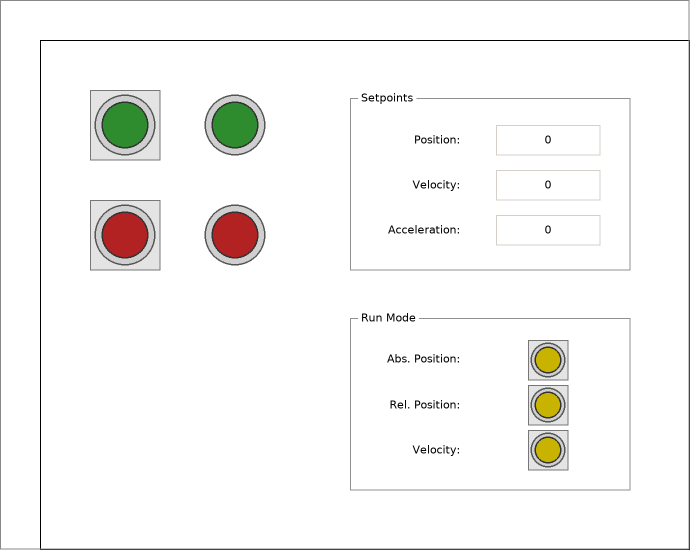
VISUALIZATION Visualization  // 690x550
    RoundedRectangle (40,40 650x510)
    PushSwitch (90,90 70x70), tooltip "START", behaviour: TOGGLE, style: Switch-PushSwitch-Green
    Lamp1 (200,90 70x70), style: Lamp-Lamp1-Green
    PushSwitch (90,200 70x70), tooltip "STOP", behaviour: TOGGLE, style: Switch-PushSwitch-Red
    Lamp1 (200,200 70x70), style: Lamp-Lamp1-Red
    GroupBox (350,90 280x180), "Setpoints"
        Label (16,80 97x30), "Velocity:"
        Label (16,125 97x30), "Acceleration:"
        Textfield (146,80 104x30), "0"
        Textfield (146,35 104x30), "0"
        Textfield (146,125 104x30), "0"
        Label (16,35 97x30), "Position:"
    GroupBox (350,310 280x180), "Run Mode"
        Label (16,80 97x30), "Rel. Position:"
        Label (16,125 97x30), "Velocity:"
        Label (16,34 97x30), "Abs. Position:"
        PushSwitch (178,30 40x40), behaviour: TOGGLE, style: Switch-PushSwitch-Yellow
        PushSwitch (178,75 40x40), behaviour: TOGGLE, style: Switch-PushSwitch-Yellow
        PushSwitch (178,120 40x40), behaviour: TOGGLE, style: Switch-PushSwitch-Yellow
END_VISUALIZATION

(* stored: Version 1.1.0.1, ProductVersion 3.1.4024.12
   Visu Visualization: Id {871559c6-b0ee-4414-8ee3-84a32fbb96ef} *)
